PROGRAM P_Set_Research_Data
VAR


END_VAR

//***********************************************************************************
//
// ETH Zürich / Robotic Fabrication Lab
// HIB C 13 / Stefano-Franscini-Platz 1
// CH-8093 Zürich
// 
// ***********************************************************************************
// 
// PROJECT     :  A061 Inline Mixer
// 
// FUNCTION    :  Set all research data for the process
// 
// AUTHOR      :  Seyma Gürel / Philippe Fleischmann
// 
// EMAIL       :  scotto@arch.ethz.ch / fleischmann@arch.ehtz.ch
// 
// Copyright   :  ETH Zürich (CH) 2021
//
// ***********************************************************************************


//
// Updating Mixer 1 max speed [°/s]
GVL_ResearchData.f_RED_Control_Speed:=720;
GVL_VAR.f_MI1_MaxSpeed:=GVL_ResearchData.f_RED_Control_Speed;

//
// Updating Acceleration Pump calibration values 
GVL_ResearchData.n_RED_Acceleration_Pump_Calibration_Speed:=32767;     // [raw date]
GVL_ResearchData.n_RED_Acceleration_Pump_Calibration_Time:=T#60000MS;   // [ms]
//GVL_ResearchData.f_RED_Acceleration_Pump_Mass:=342.0;                    // [g/min]
GVL_ResearchData.f_RED_Acceleration_Pump_Density:=2.047;               // [g/ml]

END_PROGRAM

(* stored: Version 1.1.0.1, ProductVersion 3.1.4024.2
   POU P_Set_Research_Data: Id {773f30f1-b7d3-4c7e-b27f-8d66212207e7}, SpecialFunc None *)
